TYPE T_PACK_Barcode : STRING(cMAX_PACKCODE_LENGHT);
END_TYPE

(* stored: Version 1.1.0.1
   DUT T_PACK_Barcode: Id {4e2e1d01-981f-49c2-8ef1-71f0e723896a} *)
